// Mitsubishi GX Works2 project: main   PLC: FX3U/FX3UC

PROGRAM MAIN
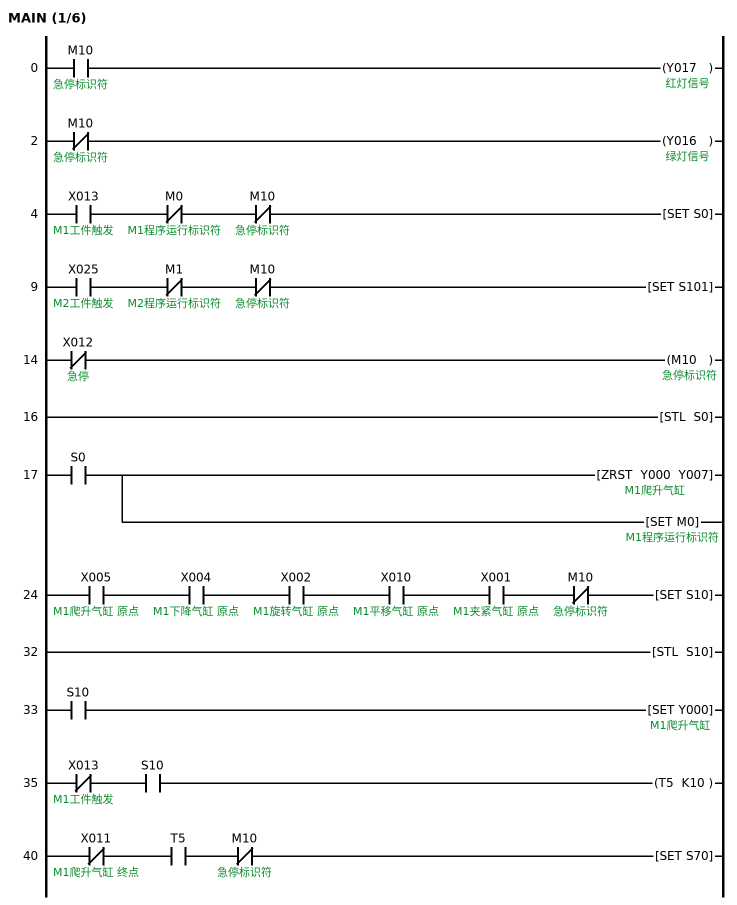
0     LD      M10  ; 急停标识符
      OUT     Y017  ; 红灯信号
2     LDI     M10  ; 急停标识符
      OUT     Y016  ; 绿灯信号
4     LD      X013  ; M1工件触发
      ANI     M0  ; M1程序运行标识符
      ANI     M10  ; 急停标识符
      SET     S0
9     LD      X025  ; M2工件触发
      ANI     M1  ; M2程序运行标识符
      ANI     M10  ; 急停标识符
      SET     S101
14    LDI     X012  ; 急停
      OUT     M10  ; 急停标识符
16    STL     S0
17    LD      S0
      ZRST    Y000 Y007  ; M1爬升气缸
      SET     M0  ; M1程序运行标识符
24    LD      X005  ; M1爬升气缸 原点
      AND     X004  ; M1下降气缸 原点
      AND     X002  ; M1旋转气缸 原点
      AND     X010  ; M1平移气缸 原点
      AND     X001  ; M1夹紧气缸 原点
      ANI     M10  ; 急停标识符
      SET     S10
32    STL     S10
33    LD      S10
      SET     Y000  ; M1爬升气缸
35    LDI     X013  ; M1工件触发
      AND     S10
      OUT     T5 K10
40    LDI     X011  ; M1爬升气缸 终点
      AND     T5
      ANI     M10  ; 急停标识符
      SET     S70
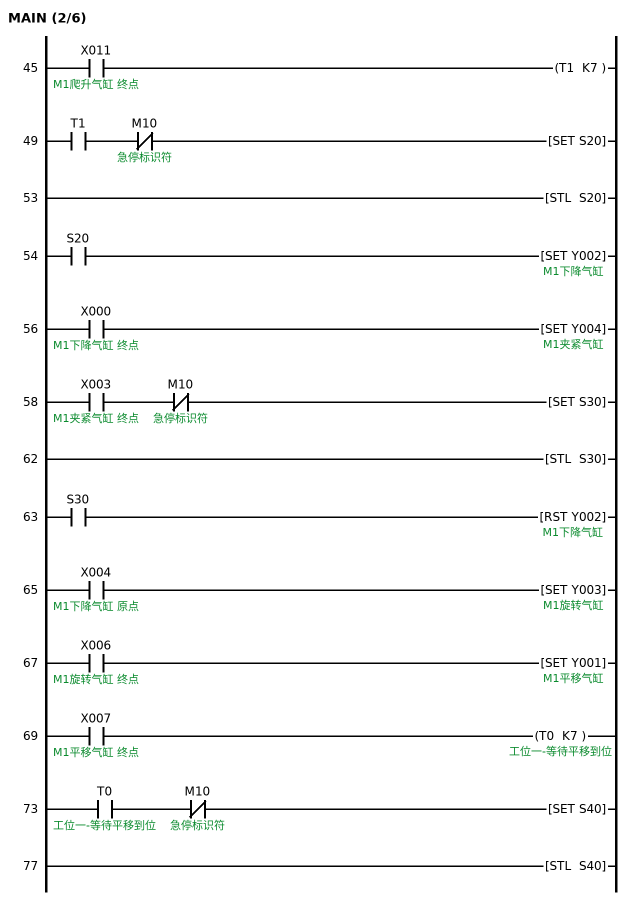
45    LD      X011  ; M1爬升气缸 终点
      OUT     T1 K7
49    LD      T1
      ANI     M10  ; 急停标识符
      SET     S20
53    STL     S20
54    LD      S20
      SET     Y002  ; M1下降气缸
56    LD      X000  ; M1下降气缸 终点
      SET     Y004  ; M1夹紧气缸
58    LD      X003  ; M1夹紧气缸 终点
      ANI     M10  ; 急停标识符
      SET     S30
62    STL     S30
63    LD      S30
      RST     Y002  ; M1下降气缸
65    LD      X004  ; M1下降气缸 原点
      SET     Y003  ; M1旋转气缸
67    LD      X006  ; M1旋转气缸 终点
      SET     Y001  ; M1平移气缸
69    LD      X007  ; M1平移气缸 终点
      OUT     T0 K7  ; 工位一-等待平移到位
73    LD      T0  ; 工位一-等待平移到位
      ANI     M10  ; 急停标识符
      SET     S40
77    STL     S40
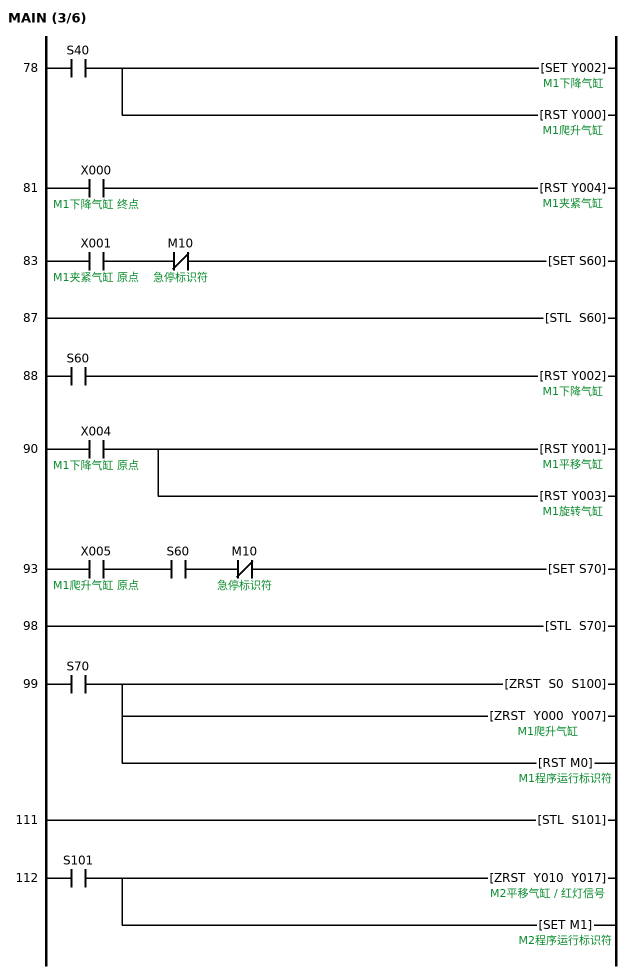
78    LD      S40
      SET     Y002  ; M1下降气缸
      RST     Y000  ; M1爬升气缸
81    LD      X000  ; M1下降气缸 终点
      RST     Y004  ; M1夹紧气缸
83    LD      X001  ; M1夹紧气缸 原点
      ANI     M10  ; 急停标识符
      SET     S60
87    STL     S60
88    LD      S60
      RST     Y002  ; M1下降气缸
90    LD      X004  ; M1下降气缸 原点
      RST     Y001  ; M1平移气缸
      RST     Y003  ; M1旋转气缸
93    LD      X005  ; M1爬升气缸 原点
      AND     S60
      ANI     M10  ; 急停标识符
      SET     S70
98    STL     S70
99    LD      S70
      ZRST    S0 S100
      ZRST    Y000 Y007
      RST     M0  ; M1程序运行标识符
111   STL     S101
112   LD      S101
      ZRST    Y010 Y017  ; M2平移气缸
      SET     M1  ; M2程序运行标识符
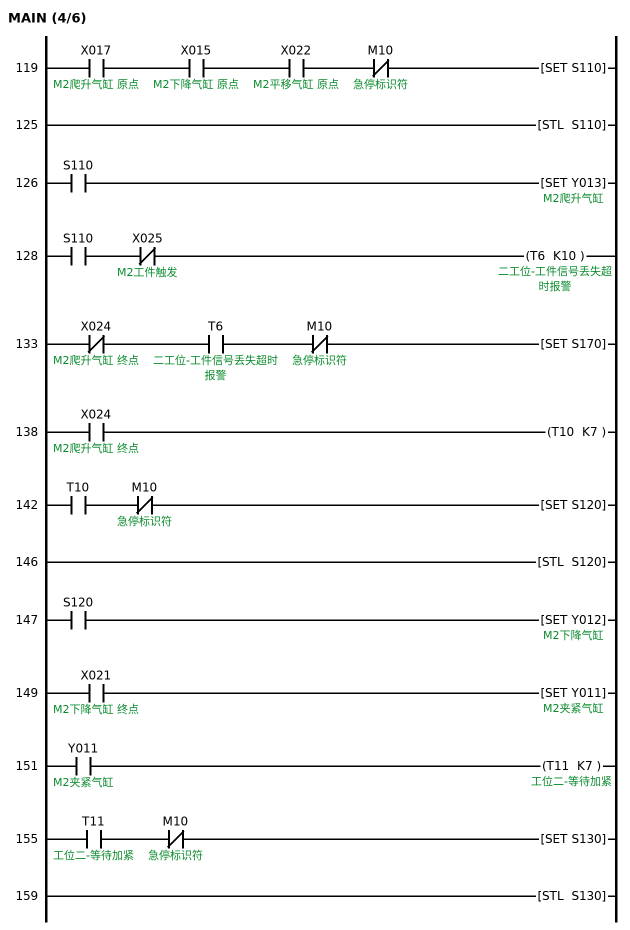
119   LD      X017  ; M2爬升气缸 原点
      AND     X015  ; M2下降气缸 原点
      AND     X022  ; M2平移气缸 原点
      ANI     M10  ; 急停标识符
      SET     S110
125   STL     S110
126   LD      S110
      SET     Y013  ; M2爬升气缸
128   LD      S110
      ANI     X025  ; M2工件触发
      OUT     T6 K10  ; 二工位-工件信号丢失超时报警
133   LDI     X024  ; M2爬升气缸 终点
      AND     T6  ; 二工位-工件信号丢失超时报警
      ANI     M10  ; 急停标识符
      SET     S170
138   LD      X024  ; M2爬升气缸 终点
      OUT     T10 K7
142   LD      T10
      ANI     M10  ; 急停标识符
      SET     S120
146   STL     S120
147   LD      S120
      SET     Y012  ; M2下降气缸
149   LD      X021  ; M2下降气缸 终点
      SET     Y011  ; M2夹紧气缸
151   LD      Y011  ; M2夹紧气缸
      OUT     T11 K7  ; 工位二-等待加紧
155   LD      T11  ; 工位二-等待加紧
      ANI     M10  ; 急停标识符
      SET     S130
159   STL     S130
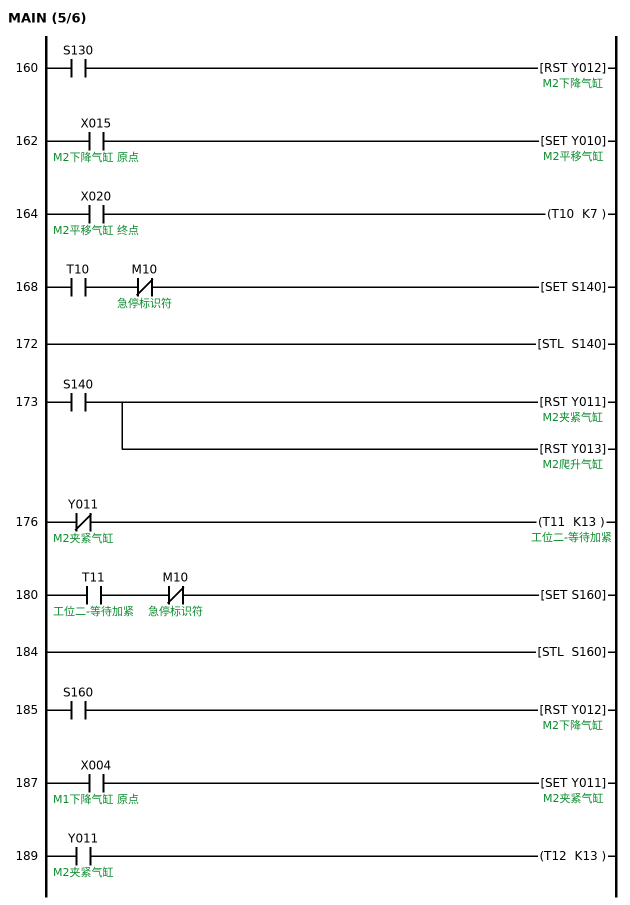
160   LD      S130
      RST     Y012  ; M2下降气缸
162   LD      X015  ; M2下降气缸 原点
      SET     Y010  ; M2平移气缸
164   LD      X020  ; M2平移气缸 终点
      OUT     T10 K7
168   LD      T10
      ANI     M10  ; 急停标识符
      SET     S140
172   STL     S140
173   LD      S140
      RST     Y011  ; M2夹紧气缸
      RST     Y013  ; M2爬升气缸
176   LDI     Y011  ; M2夹紧气缸
      OUT     T11 K13  ; 工位二-等待加紧
180   LD      T11  ; 工位二-等待加紧
      ANI     M10  ; 急停标识符
      SET     S160
184   STL     S160
185   LD      S160
      RST     Y012  ; M2下降气缸
187   LD      X004  ; M1下降气缸 原点
      SET     Y011  ; M2夹紧气缸
189   LD      Y011  ; M2夹紧气缸
      OUT     T12 K13
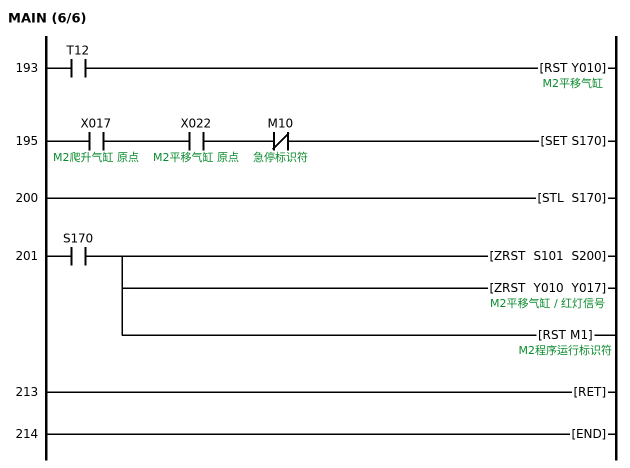
193   LD      T12
      RST     Y010  ; M2平移气缸
195   LD      X017  ; M2爬升气缸 原点
      AND     X022  ; M2平移气缸 原点
      ANI     M10  ; 急停标识符
      SET     S170
200   STL     S170
201   LD      S170
      ZRST    S101 S200
      ZRST    Y010 Y017
      RST     M1  ; M2程序运行标识符
213   RET
214   END
END_PROGRAM
